{attribute 'GeneratedUsingTerminal: EL4011-0000-0016'}
{attribute addProperty BoxType "EL4011-0000-0016"}
{attribute addProperty Id "AO_OutputsAT %Q*AO_Output_Channel_BA7EBB7C2WcStateAT %I*WcState_0B2B16F91InfoDataAT %I*InfoData_94A18F5E2"}
{attribute addProperty CRC "801311827"}
{attribute addProperty Size "5"}
TYPE EL4011_2FC30C53 EXTENDS EtcSlaveTerminalBase_947E5A46 :
STRUCT
	{attribute addProperty Name "AO_Outputs"}
	AO_Outputs : AO_Output_Channel_BA7EBB7C;
	{attribute addProperty Name "WcState"}
	WcState : WcState_0B2B16F9;
	{attribute addProperty Name "InfoData"}
	InfoData : InfoData_94A18F5E;
END_STRUCT
END_TYPE

(* stored: Version 1.2.0.0, ProductVersion 3.1.4024.9
   DUT EL4011_2FC30C53: Id {4227a932-69b8-4bb9-8a3c-442b54a964c8} *)
